// TIA Portal V17 export
// export: Created 2024-01-30T08:49:16.0849601Z, ExportSetting WithDefaults, DisplayName Totally Integrated Automation Portal, DisplayVersion V17 Update 6, DisplayName TIA Portal Openness, DisplayVersion V17 Update 6, DisplayName TIA Portal Version Control Interface, DisplayVersion V17, DisplayName STEP 7 Professional, DisplayVersion V17 Update 6, DisplayName STEP 7 Safety, DisplayVersion V17 Update 6, DisplayName WinCC Advanced, DisplayVersion V17 Update 6
DATA_BLOCK "DATA_LOGGING"   // DB25
{ S7_Optimized_Access := 'TRUE' }
VERSION : 0.1
// stored: AutoNumber true, DBAccessibleFromOPCUA true, DBAccessibleFromWebserver true, IsOnlyStoredInLoadMemory false, IsRetainMemResEnabled false, IsWriteProtectedInAS false, MemoryReserve 100
   VAR
      Record : UDInt;
      "Name" : String := 'Logging';
      ID : DWord := 1;
      Header : String := 'A350-1000, Errors';
      Data : Struct
         First : UDInt;
         Second : UDInt;
         Third : UDInt;
      END_STRUCT;
   END_VAR
BEGIN
END_DATA_BLOCK
